% RSLogix 500 project PUMP_PROTECTION.RSS, saved by version 8.30.00.16 %
PROJECT "UNTITLED"    % processor: Bul.1763 MicroLogix 1100 Series B %

PROGRAM FILES
  LAD 2 "MAIN"  5 rungs
  LAD 3 "IO"  11 rungs
  LAD 4 "CTRL"  12 rungs
  LAD 5 "ALARMS"  11 rungs
  LAD 6 "HOA"  9 rungs

DATA FILES
  O0 OUTPUT  4 elements
  I1 INPUT  6 elements
  S2 STATUS  66 elements
  B3 BINARY  2 elements
  T4 TIMER  4 elements
  C5 COUNTER  1 elements
  R6 CONTROL  1 elements
  N7 INTEGER  5 elements
  F8 FLOAT  1 elements

LADDER 2 "MAIN"
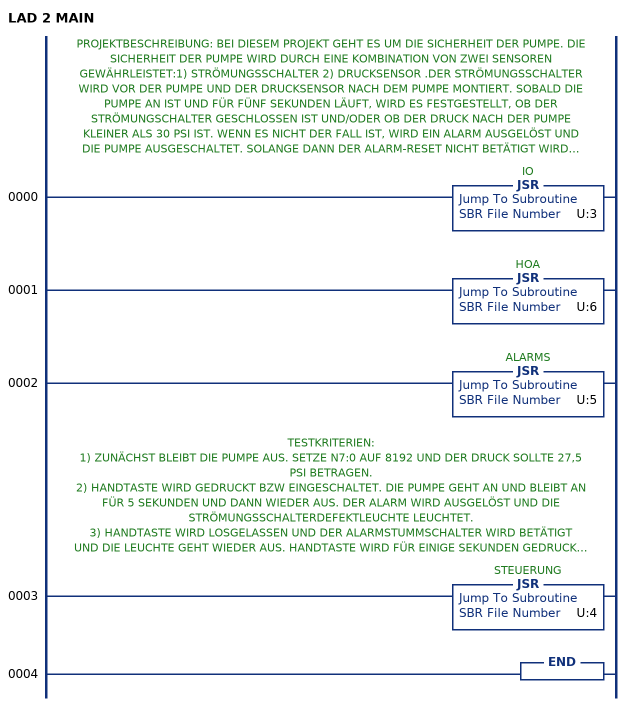
% Rung: 0 %
% PROJEKTBESCHREIBUNG: BEI DIESEM PROJEKT GEHT ES UM DIE SICHERHEIT DER PUMPE. DIE SICHERHEIT DER PUMPE WIRD DURCH EINE KOMBINATION VON ZWEI SENSOREN GEWÄHRLEISTET:1) STRÖMUNGSSCHALTER 2) DRUCKSENSOR .DER STRÖMUNGSSCHALTER WIRD VOR DER PUMPE UND DER DRUCKSENSOR NACH DEM PUMPE MONTIERT. SOBALD DIE PUMPE AN IST UND FÜR FÜNF SEKUNDEN LÄUFT, WIRD ES FESTGESTELLT, OB DER STRÖMUNGSCHALTER GESCHLOSSEN IST UND/ODER OB DER DRUCK NACH DER PUMPE KLEINER ALS 30 PSI IST. WENN ES NICHT DER FALL IST, WIRD EIN ALARM AUSGELÖST UND DIE PUMPE AUSGESCHALTET. SOLANGE DANN DER ALARM-RESET NICHT BETÄTIGT WIRD, KANN DIE PUMPE NICHT WIEDER IM BETRIEB GENOMMEN WERDEN. AUßERDEM WIRD DIE PUMP MITTELS HAND/AUTOMATIK/AUS SCHALTER BETRIEBEN. SOLANGE DIE HANDTASTE GEDRUCKT BLEIBT, LÄUFT DIE PUMPE. SOBALD DIE HANDTASTE LOSGELASSEN WIRD GEHT DIE PUMPE WIRD IM MODUS, DAS VOR DEM HAND-MODUS AKTIV WAR. IN AUTO-MODUS LÄUFT DIE PUMPE IN EINEM ZYKLUS. DAS HEIßT, DIE PUMPE IST FÜR 30 SEKUNDEN AN UND DANN BLEIBT AUS FÜR 10 SEKUNDEN UND DANN WIEDER AN FÜR 30 SEKUNDEN UND SO WEITER. IM OFF-MODUS (AUS) BLEIBT DIE PUMPE AUS. FOLGEND SIND DIE IO FÜR DAS PROGRAMM:
% 1) I:0/0 - STRÖMUNGSCHALTER
% 2) I:0/1 - ALARM-RESET
% 3) I:0/2 - ALARMSTUMMSCHALTER
% 4)  I:0/3 - HANDTASTE
% 5)  I:0/4 - OFFTASTE
% 6)  I:0/5 - AUTOTASTE
% 7) N7:0 - DRUCKSENSOR (0-16383) DA DIESES PROGRAMM AUF EMULATE GETESTET WURDE, WURDE DER SENSOR DURCH EINE INTEGER ERSETZT.
% 8) O:0/0 - PUMPE
% 9) O:0/1 -STTRÖMUNGSSCHALTERDEFEKTLEUCHTE
% 10) O:0/2 - DRUCKSENSORDEFEKTLEUCHTE %
SOR JSR U:3 EOR
%   U:3  "IO" %
% Rung: 1 %
SOR JSR U:6 EOR
%   U:6  "HOA" %
% Rung: 2 %
SOR JSR U:5 EOR
%   U:5  "ALARMS" %
% Rung: 3 %
% TESTKRITERIEN:
% 1) ZUNÄCHST BLEIBT DIE PUMPE AUS. SETZE N7:0 AUF 8192 UND DER DRUCK SOLLTE 27,5 PSI BETRAGEN.
% 2) HANDTASTE WIRD GEDRUCKT BZW EINGESCHALTET. DIE PUMPE GEHT AN UND BLEIBT AN FÜR 5 SEKUNDEN UND DANN WIEDER AUS. DER ALARM WIRD AUSGELÖST UND DIE STRÖMUNGSSCHALTERDEFEKTLEUCHTE LEUCHTET.
% 3) HANDTASTE WIRD LOSGELASSEN UND DER ALARMSTUMMSCHALTER WIRD BETÄTIGT UND DIE LEUCHTE GEHT WIEDER AUS. HANDTASTE WIRD FÜR EINIGE SEKUNDEN GEDRUCKT UND WIEDER LOSGELASSEN ABER DIE PUMPE GEHT NICHT AN.
% 4) AUTOTASTE WIRD GETOGGELT. DIE PUMPEZYKLUS SOLLTE NICHT AN GEHEN
% 5) ALARMRESET WIRD BETÄTIGT UND DANN WIRD STRÖMUNGSCHALTER GESCHALTET. NUN WIRD AUTOTASTE GETOGGELT. DIE PUMPE SOLLTE IM ZYKLUS LAUFEN.
% 6) NUN WIRD HANDTASTE GEDRUCKT FÜR UNGEFÄHR 20 SEKUNDEN. DIE PUMPE SOLLTE AUS DEM ZYKLUS RAUS UND STÄNDIG LAUFEN. WIRD DIE HANDTASTE WIEDER GELASSEN SOLLTE DIE PUMPE WIRD IM ZYKLUS LAUFEN.
% 7) SETZE N7:0 AUF 10000 UND DIE PUMPE SOLLTE NACH 5 SEKUNDEN AUS GEHEN. DER ALARM WIRD AUSGELÖST UND DIE DRUCKSENSORDEFEKTLEUCHTE LEUCHTET. DER DRUCKWERT BETRÄGT 33,5 PSI. %
SOR JSR U:4 EOR
%   U:4  "STEUERUNG" %
% Rung: 4 %
SOR END EOR

LADDER 3 "IO"
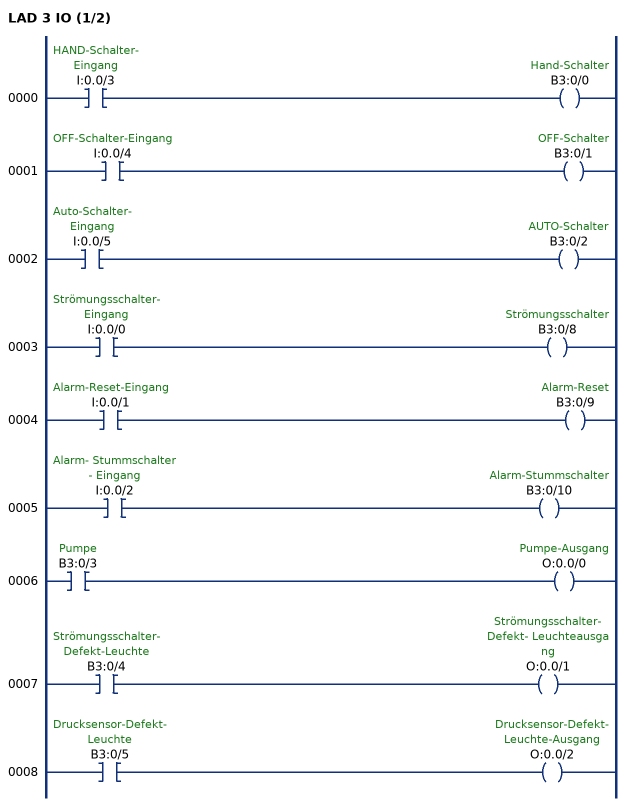
% Rung: 0 %
SOR XIC I:0.0/3 OTE B3:0/0 EOR
%   I:0.0/3  "HAND-Schalter- Eingang" %
%   B3:0/0  "Hand-Schalter" %
% Rung: 1 %
SOR XIC I:0.0/4 OTE B3:0/1 EOR
%   I:0.0/4  "OFF-Schalter-Eingang" %
%   B3:0/1  "OFF-Schalter" %
% Rung: 2 %
SOR XIC I:0.0/5 OTE B3:0/2 EOR
%   I:0.0/5  "Auto-Schalter- Eingang" %
%   B3:0/2  "AUTO-Schalter" %
% Rung: 3 %
SOR XIC I:0.0/0 OTE B3:0/8 EOR
%   I:0.0/0  "Strömungsschalter- Eingang" %
%   B3:0/8  "Strömungsschalter" %
% Rung: 4 %
SOR XIC I:0.0/1 OTE B3:0/9 EOR
%   I:0.0/1  "Alarm-Reset-Eingang" %
%   B3:0/9  "Alarm-Reset" %
% Rung: 5 %
SOR XIC I:0.0/2 OTE B3:0/10 EOR
%   I:0.0/2  "Alarm- Stummschalter- Eingang" %
%   B3:0/10  "Alarm-Stummschalter" %
% Rung: 6 %
SOR XIC B3:0/3 OTE O:0.0/0 EOR
%   B3:0/3  "Pumpe" %
%   O:0.0/0  "Pumpe-Ausgang" %
% Rung: 7 %
SOR XIC B3:0/4 OTE O:0.0/1 EOR
%   B3:0/4  "Strömungsschalter- Defekt-Leuchte" %
%   O:0.0/1  "Strömungsschalter- Defekt- Leuchteausgang" %
% Rung: 8 %
SOR XIC B3:0/5 OTE O:0.0/2 EOR
%   B3:0/5  "Drucksensor-Defekt- Leuchte" %
%   O:0.0/2  "Drucksensor-Defekt- Leuchte-Ausgang" %

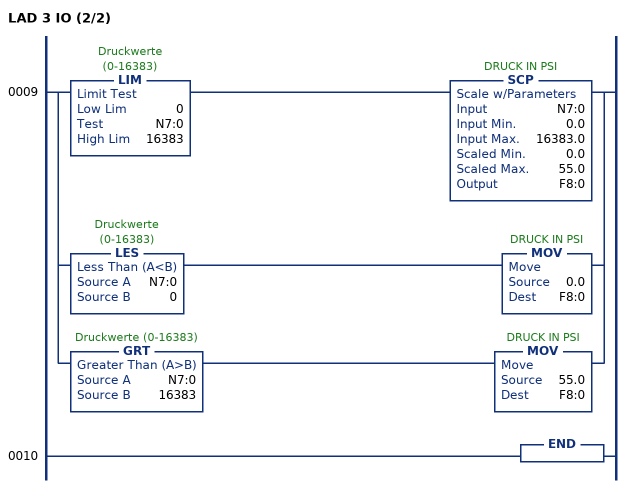
% Rung: 9 %
SOR BST LIM 0 N7:0 16383 SCP N7:0 0.0 16383.0 0.0 55.0 F8:0 NXB LES N7:0 0 MOV 0.0 F8:0 NXB GRT N7:0 16383 MOV 55.0 F8:0 BND EOR
%   N7:0  "Druckwerte (0-16383)" %
%   F8:0  "DRUCK IN PSI" %
% Rung: 10 %
SOR END EOR

LADDER 4 "CTRL"
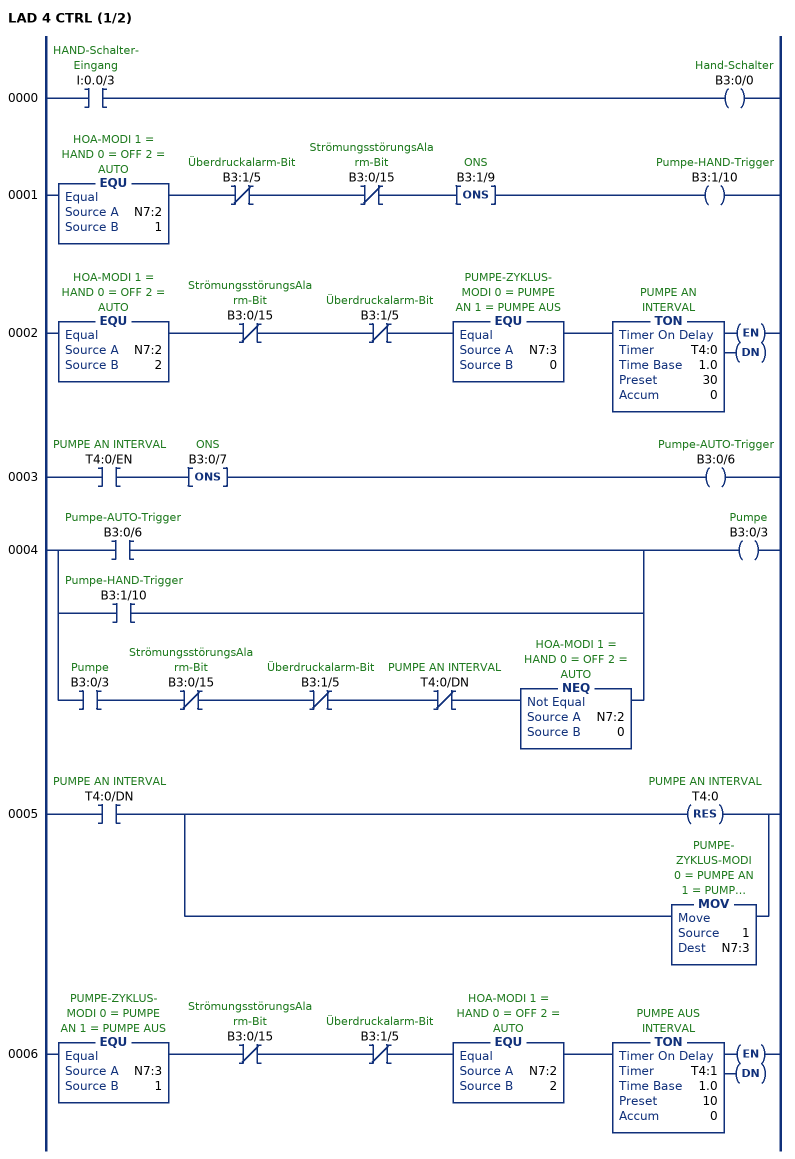
% Rung: 0 %
SOR XIC I:0.0/3 OTE B3:0/0 EOR
%   I:0.0/3  "HAND-Schalter- Eingang" %
%   B3:0/0  "Hand-Schalter" %
% Rung: 1 %
SOR EQU N7:2 1 XIO B3:1/5 XIO B3:0/15 ONS B3:1/9 OTE B3:1/10 EOR
%   N7:2  "HOA-MODI 1 = HAND 0 = OFF 2 = AUTO" %
%   B3:1/5  "Überdruckalarm-Bit" %
%   B3:0/15  "StrömungsstörungsAla rm-Bit" %
%   B3:1/9  "ONS" %
%   B3:1/10  "Pumpe-HAND-Trigger" %
% Rung: 2 %
SOR EQU N7:2 2 XIO B3:0/15 XIO B3:1/5 EQU N7:3 0 TON T4:0 1.0 30 0 EOR
%   N7:2  "HOA-MODI 1 = HAND 0 = OFF 2 = AUTO" %
%   B3:0/15  "StrömungsstörungsAla rm-Bit" %
%   B3:1/5  "Überdruckalarm-Bit" %
%   N7:3  "PUMPE-ZYKLUS-MODI 0 = PUMPE AN 1 = PUMPE AUS" %
%   T4:0  "PUMPE AN INTERVAL" %
% Rung: 3 %
SOR XIC T4:0/EN ONS B3:0/7 OTE B3:0/6 EOR
%   T4:0  "PUMPE AN INTERVAL" %
%   B3:0/7  "ONS" %
%   B3:0/6  "Pumpe-AUTO-Trigger" %
% Rung: 4 %
SOR BST BST XIC B3:0/6 NXB XIC B3:1/10 BND NXB XIC B3:0/3 XIO B3:0/15 XIO B3:1/5 XIO T4:0/DN NEQ N7:2 0 BND OTE B3:0/3 EOR
%   B3:0/6  "Pumpe-AUTO-Trigger" %
%   B3:1/10  "Pumpe-HAND-Trigger" %
%   B3:0/3  "Pumpe" %
%   B3:0/15  "StrömungsstörungsAla rm-Bit" %
%   B3:1/5  "Überdruckalarm-Bit" %
%   T4:0  "PUMPE AN INTERVAL" %
%   N7:2  "HOA-MODI 1 = HAND 0 = OFF 2 = AUTO" %
% Rung: 5 %
SOR XIC T4:0/DN BST RES T4:0 NXB MOV 1 N7:3 BND EOR
%   T4:0  "PUMPE AN INTERVAL" %
%   N7:3  "PUMPE-ZYKLUS-MODI 0 = PUMPE AN 1 = PUMPE AUS" %
% Rung: 6 %
SOR EQU N7:3 1 XIO B3:0/15 XIO B3:1/5 EQU N7:2 2 TON T4:1 1.0 10 0 EOR
%   N7:3  "PUMPE-ZYKLUS-MODI 0 = PUMPE AN 1 = PUMPE AUS" %
%   B3:0/15  "StrömungsstörungsAla rm-Bit" %
%   B3:1/5  "Überdruckalarm-Bit" %
%   N7:2  "HOA-MODI 1 = HAND 0 = OFF 2 = AUTO" %
%   T4:1  "PUMPE AUS INTERVAL" %

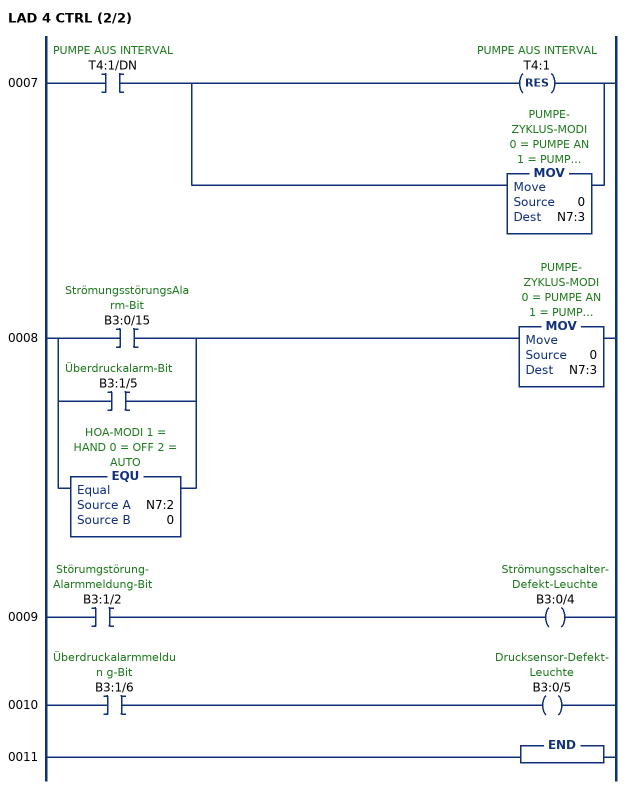
% Rung: 7 %
SOR XIC T4:1/DN BST RES T4:1 NXB MOV 0 N7:3 BND EOR
%   T4:1  "PUMPE AUS INTERVAL" %
%   N7:3  "PUMPE-ZYKLUS-MODI 0 = PUMPE AN 1 = PUMPE AUS" %
% Rung: 8 %
SOR BST XIC B3:0/15 NXB XIC B3:1/5 NXB EQU N7:2 0 BND MOV 0 N7:3 EOR
%   B3:0/15  "StrömungsstörungsAla rm-Bit" %
%   B3:1/5  "Überdruckalarm-Bit" %
%   N7:2  "HOA-MODI 1 = HAND 0 = OFF 2 = AUTO" %
%   N7:3  "PUMPE-ZYKLUS-MODI 0 = PUMPE AN 1 = PUMPE AUS" %
% Rung: 9 %
SOR XIC B3:1/2 OTE B3:0/4 EOR
%   B3:1/2  "Störumgstörung- Alarmmeldung-Bit" %
%   B3:0/4  "Strömungsschalter- Defekt-Leuchte" %
% Rung: 10 %
SOR XIC B3:1/6 OTE B3:0/5 EOR
%   B3:1/6  "Überdruckalarmmeldun g-Bit" %
%   B3:0/5  "Drucksensor-Defekt- Leuchte" %
% Rung: 11 %
SOR END EOR

LADDER 5 "ALARMS"
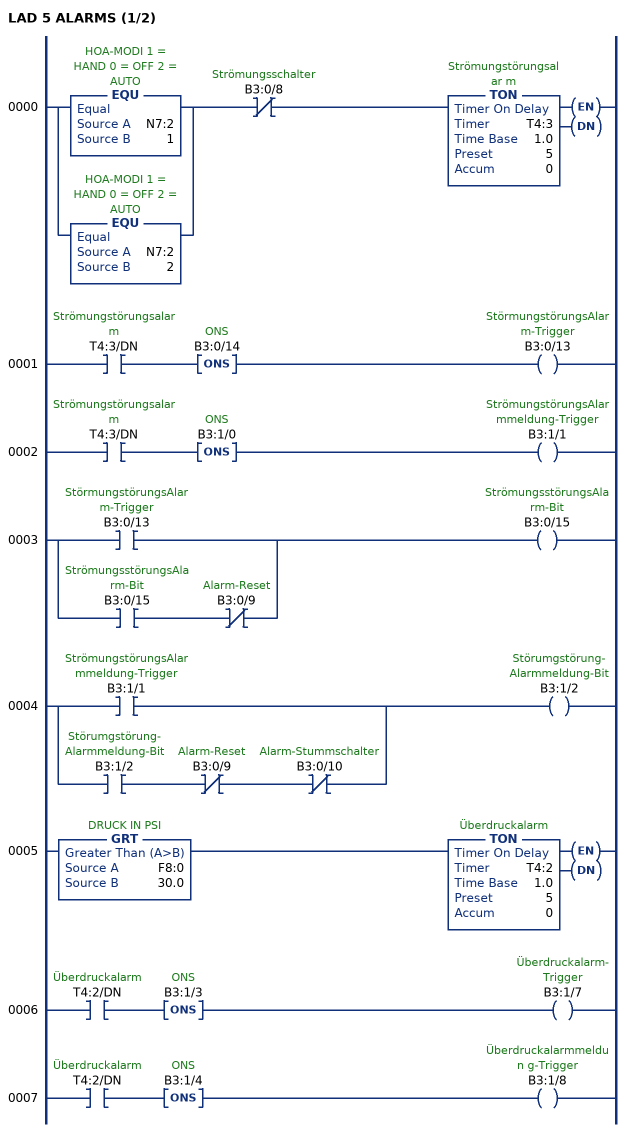
% Rung: 0 %
SOR BST EQU N7:2 1 NXB EQU N7:2 2 BND XIO B3:0/8 TON T4:3 1.0 5 0 EOR
%   N7:2  "HOA-MODI 1 = HAND 0 = OFF 2 = AUTO" %
%   B3:0/8  "Strömungsschalter" %
%   T4:3  "Strömungstörungsalar m" %
% Rung: 1 %
SOR XIC T4:3/DN ONS B3:0/14 OTE B3:0/13 EOR
%   T4:3  "Strömungstörungsalar m" %
%   B3:0/14  "ONS" %
%   B3:0/13  "StörmungstörungsAlar m-Trigger" %
% Rung: 2 %
SOR XIC T4:3/DN ONS B3:1/0 OTE B3:1/1 EOR
%   T4:3  "Strömungstörungsalar m" %
%   B3:1/0  "ONS" %
%   B3:1/1  "StrömungstörungsAlar mmeldung-Trigger" %
% Rung: 3 %
SOR BST XIC B3:0/13 NXB XIC B3:0/15 XIO B3:0/9 BND OTE B3:0/15 EOR
%   B3:0/13  "StörmungstörungsAlar m-Trigger" %
%   B3:0/15  "StrömungsstörungsAla rm-Bit" %
%   B3:0/9  "Alarm-Reset" %
% Rung: 4 %
SOR BST XIC B3:1/1 NXB XIC B3:1/2 XIO B3:0/9 XIO B3:0/10 BND OTE B3:1/2 EOR
%   B3:1/1  "StrömungstörungsAlar mmeldung-Trigger" %
%   B3:1/2  "Störumgstörung- Alarmmeldung-Bit" %
%   B3:0/9  "Alarm-Reset" %
%   B3:0/10  "Alarm-Stummschalter" %
% Rung: 5 %
SOR GRT F8:0 30.0 TON T4:2 1.0 5 0 EOR
%   F8:0  "DRUCK IN PSI" %
%   T4:2  "Überdruckalarm" %
% Rung: 6 %
SOR XIC T4:2/DN ONS B3:1/3 OTE B3:1/7 EOR
%   T4:2  "Überdruckalarm" %
%   B3:1/3  "ONS" %
%   B3:1/7  "Überdruckalarm- Trigger" %
% Rung: 7 %
SOR XIC T4:2/DN ONS B3:1/4 OTE B3:1/8 EOR
%   T4:2  "Überdruckalarm" %
%   B3:1/4  "ONS" %
%   B3:1/8  "Überdruckalarmmeldun g-Trigger" %

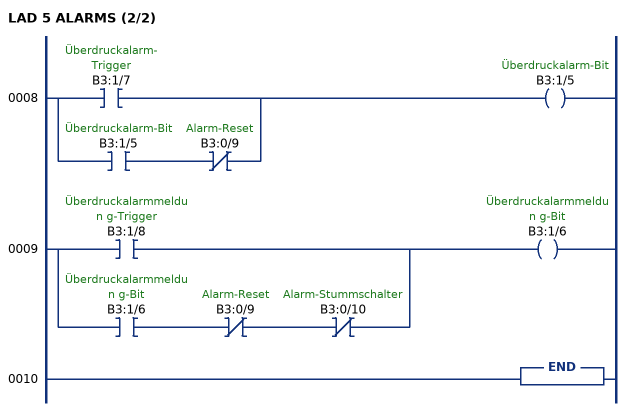
% Rung: 8 %
SOR BST XIC B3:1/7 NXB XIC B3:1/5 XIO B3:0/9 BND OTE B3:1/5 EOR
%   B3:1/7  "Überdruckalarm- Trigger" %
%   B3:1/5  "Überdruckalarm-Bit" %
%   B3:0/9  "Alarm-Reset" %
% Rung: 9 %
SOR BST XIC B3:1/8 NXB XIC B3:1/6 XIO B3:0/9 XIO B3:0/10 BND OTE B3:1/6 EOR
%   B3:1/8  "Überdruckalarmmeldun g-Trigger" %
%   B3:1/6  "Überdruckalarmmeldun g-Bit" %
%   B3:0/9  "Alarm-Reset" %
%   B3:0/10  "Alarm-Stummschalter" %
% Rung: 10 %
SOR END EOR

LADDER 6 "HOA"
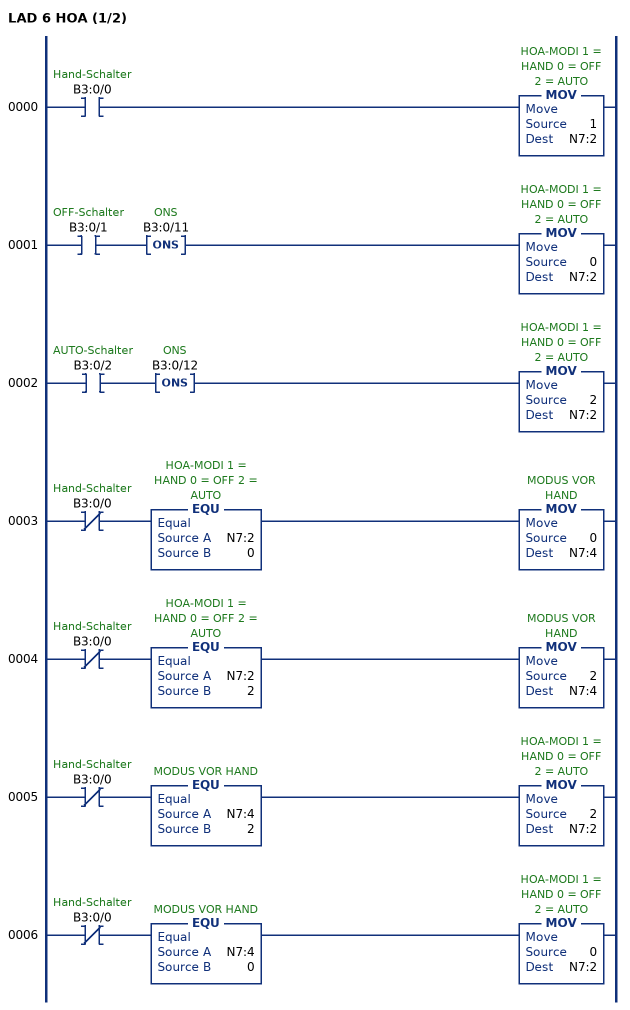
% Rung: 0 %
SOR XIC B3:0/0 MOV 1 N7:2 EOR
%   B3:0/0  "Hand-Schalter" %
%   N7:2  "HOA-MODI 1 = HAND 0 = OFF 2 = AUTO" %
% Rung: 1 %
SOR XIC B3:0/1 ONS B3:0/11 MOV 0 N7:2 EOR
%   B3:0/1  "OFF-Schalter" %
%   B3:0/11  "ONS" %
%   N7:2  "HOA-MODI 1 = HAND 0 = OFF 2 = AUTO" %
% Rung: 2 %
SOR XIC B3:0/2 ONS B3:0/12 MOV 2 N7:2 EOR
%   B3:0/2  "AUTO-Schalter" %
%   B3:0/12  "ONS" %
%   N7:2  "HOA-MODI 1 = HAND 0 = OFF 2 = AUTO" %
% Rung: 3 %
SOR XIO B3:0/0 EQU N7:2 0 MOV 0 N7:4 EOR
%   B3:0/0  "Hand-Schalter" %
%   N7:2  "HOA-MODI 1 = HAND 0 = OFF 2 = AUTO" %
%   N7:4  "MODUS VOR HAND" %
% Rung: 4 %
SOR XIO B3:0/0 EQU N7:2 2 MOV 2 N7:4 EOR
%   B3:0/0  "Hand-Schalter" %
%   N7:2  "HOA-MODI 1 = HAND 0 = OFF 2 = AUTO" %
%   N7:4  "MODUS VOR HAND" %
% Rung: 5 %
SOR XIO B3:0/0 EQU N7:4 2 MOV 2 N7:2 EOR
%   B3:0/0  "Hand-Schalter" %
%   N7:4  "MODUS VOR HAND" %
%   N7:2  "HOA-MODI 1 = HAND 0 = OFF 2 = AUTO" %
% Rung: 6 %
SOR XIO B3:0/0 EQU N7:4 0 MOV 0 N7:2 EOR
%   B3:0/0  "Hand-Schalter" %
%   N7:4  "MODUS VOR HAND" %
%   N7:2  "HOA-MODI 1 = HAND 0 = OFF 2 = AUTO" %

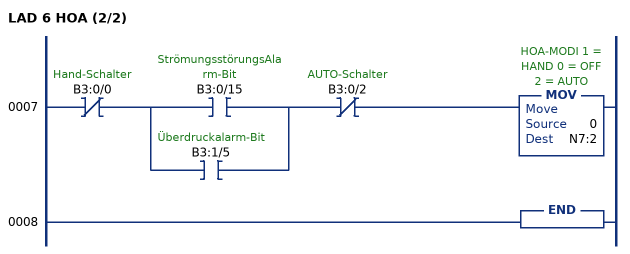
% Rung: 7 %
SOR XIO B3:0/0 BST XIC B3:0/15 NXB XIC B3:1/5 BND XIO B3:0/2 MOV 0 N7:2 EOR
%   B3:0/0  "Hand-Schalter" %
%   B3:0/15  "StrömungsstörungsAla rm-Bit" %
%   B3:1/5  "Überdruckalarm-Bit" %
%   B3:0/2  "AUTO-Schalter" %
%   N7:2  "HOA-MODI 1 = HAND 0 = OFF 2 = AUTO" %
% Rung: 8 %
SOR END EOR

OTHER DOCUMENTED ADDRESSES
  N7:1  "Druck in Psi"
  T4:4  "Überdruckalarm"

DATA TABLE (non-zero values as saved)
DATA T4
% .PRE .ACC %
% T4:0 % 30 0
% T4:1 % 10 0
% T4:2 % 5 0
% T4:3 % 5 0
